// TIA Portal V19 export
FUNCTION_BLOCK "MWhell_Check"   // FB134, LAD
// stored: MemoryReserve 100, SetENOAutomatically false
   VAR_INPUT
      MWheel_Sensor { ExternalAccessible := 'False'; ExternalVisible := 'False'; ExternalWritable := 'False'} : Int;
      MaterialPresence : Bool;
   END_VAR
   VAR_OUTPUT
      CheckOK : Bool;
      ParameterError : Bool;
      GearRatioError : Bool;
      WheelMoving : Bool;
      LeadScrewErr { ExternalAccessible := 'False'; ExternalVisible := 'False'; ExternalWritable := 'False'} : LReal;
      CalculatedLeadScrew { ExternalAccessible := 'False'; ExternalVisible := 'False'; ExternalWritable := 'False'} : LReal;
   END_VAR
   VAR_IN_OUT
      TO_Ax : TO_PositioningAxis;
   END_VAR
   VAR
      tCheck : IEC_TIMER;
   END_VAR
BEGIN

REGION Network 1 (SCL)
   #ParameterError :=  (#TO_Ax.LoadGear.Numerator = 0.0 )
                   OR (#TO_Ax.LoadGear.Denominator = 0.0)
                   OR (#TO_Ax.Mechanics.LeadScrew = 0.0);

   IF #ParameterError THEN
       ENO := #CheckOK := FALSE;
       RETURN;
   END_IF;
END_REGION

REGION Network 2 (SCL): Velocity too low for calculation
   IF #TO_Ax.Velocity < #TO_Ax.StandstillSignal.VelocityThreshold THEN
       #WheelMoving    := FALSE;
       ENO := #CheckOK;
       RETURN;
   END_IF;
END_REGION

REGION Network 3 (SCL): LeadScrew calculated and error
   #CalculatedLeadScrew := (#TO_Ax.StatusSensor[#MWheel_Sensor].Velocity * UDINT_TO_LREAL(#TO_Ax.LoadGear.Numerator))
                         / (#TO_Ax.ActualSpeed * UDINT_TO_LREAL(#TO_Ax.LoadGear.Denominator));



   CASE #TO_Ax.Units.VelocityUnit OF
       1061: (* m/s *)     #CalculatedLeadScrew := #CalculatedLeadScrew * 60000.0;            
       1524: (* mm/min *) ;     
       1525: (* m/min *)   #CalculatedLeadScrew := #CalculatedLeadScrew * 1000.0;
   END_CASE;

   #LeadScrewErr   := 100.0 * (#TO_Ax.Mechanics.LeadScrew - #CalculatedLeadScrew) / #TO_Ax.Mechanics.LeadScrew;
END_REGION

REGION Network 4 (SCL): Wheel moving / Gear ratio Error
   #WheelMoving    := #TO_Ax.StatusSensor[#MWheel_Sensor].Velocity > #TO_Ax.StandstillSignal.VelocityThreshold;
   #GearRatioError := ABS(#LeadScrewErr) > 10.0 AND #WheelMoving;
END_REGION

REGION Network 5
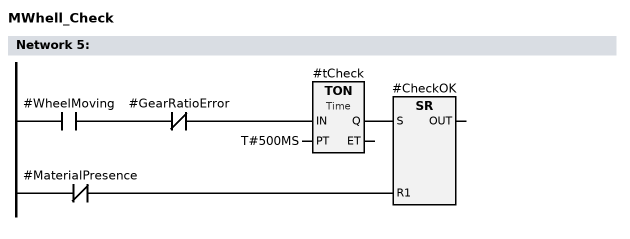
   RUNG wire#powerrail
      Contact( #WheelMoving )
      I_Contact( #GearRatioError )
      { S7_Templates := "time_type := Time" } #tCheck.TON(pt := T#500MS, et =>)
      S_SR(operand := #CheckOK, r1 := wire#w1)
   END_RUNG
   RUNG wire#powerrail
      I_Contact( #MaterialPresence )
   END_RUNG wire#w1
   // the same network as SCL:
   #tCheck.TON(IN := #WheelMoving AND NOT #GearRatioError, PT := T#500MS);
   IF #tCheck.Q THEN
       #CheckOK := TRUE;   // SR flip-flop
   END_IF;
   IF NOT #MaterialPresence THEN #CheckOK := FALSE; END_IF;
END_REGION

REGION Network 6 (SCL): ENO
   ENO := #CheckOK;
END_REGION
END_FUNCTION_BLOCK
